TYPE "MEStoPLC_ResultsStoredScanExchange_ext"
VERSION : 0.1
   STRUCT
      Load_ResultsStored1OK : Bool;
      Load_ResultsStored1NG : Bool;
      Load_ResultsStored1ReqMesDone : Bool;
      Load_ResultsStored1Spare : Bool;
      Load_ResultsStored1Spare1 : Bool;
      Load_ResultsStored1Spare2 : Bool;
      Load_ResultsStored1Spare3 : Bool;
      Load_ResultsStored1Spare4 : Bool;
      Load_ResultsStored2OK : Bool;
      Load_ResultsStored2NG : Bool;
      Load_ResultsStored2ReqMesDone : Bool;
      Load_ResultsStored2Spare : Bool;
      Load_ResultsStored2Spare1 : Bool;
      Load_ResultsStored2Spare2 : Bool;
      Load_ResultsStored2Spare3 : Bool;
      Load_ResultsStored2Spare4 : Bool;
      Load_ResultsStored3OK : Bool;
      Load_ResultsStored3NG : Bool;
      Load_ResultsStored3ReqMesDone : Bool;
      Load_ResultsStored3Spare : Bool;
      Load_ResultsStored3Spare1 : Bool;
      Load_ResultsStored3Spare2 : Bool;
      Load_ResultsStored3Spare3 : Bool;
      Load_ResultsStored3Spare4 : Bool;
      Load_ResultsStored4OK : Bool;
      Load_ResultsStored4NG : Bool;
      Load_ResultsStored4ReqMesDone : Bool;
      Load_ResultsStored4Spare : Bool;
      Load_ResultsStored4Spare1 : Bool;
      Load_ResultsStored4Spare2 : Bool;
      Load_ResultsStored4Spare3 : Bool;
      Load_ResultsStored4Spare4 : Bool;
      Load_ResultsStored5OK : Bool;
      Load_ResultsStored5NG : Bool;
      Load_ResultsStored5ReqMesDone : Bool;
      Load_ResultsStored5Spare : Bool;
      Load_ResultsStored5Spare1 : Bool;
      Load_ResultsStored5Spare2 : Bool;
      Load_ResultsStored5Spare3 : Bool;
      Load_ResultsStored5Spare4 : Bool;
      Load_ResultsStored6OK : Bool;
      Load_ResultsStored6NG : Bool;
      Load_ResultsStored6ReqMesDone : Bool;
      Load_ResultsStored6Spare : Bool;
      Load_ResultsStored6Spare1 : Bool;
      Load_ResultsStored6Spare2 : Bool;
      Load_ResultsStored6Spare3 : Bool;
      Load_ResultsStored6Spare4 : Bool;
      Spare : Byte;
      Load_ResultsStored7OK : Bool;
      Load_ResultsStored7NG : Bool;
      Load_ResultsStored7ReqMesDone : Bool;
      Load_ResultsStored7Spare : Bool;
      Load_ResultsStored7Spare1 : Bool;
      Load_ResultsStored7Spare2 : Bool;
      Load_ResultsStored7Spare3 : Bool;
      Load_ResultsStored7Spare4 : Bool;
      Load_ResultsStored8OK : Bool;
      Load_ResultsStored8NG : Bool;
      Load_ResultsStored8ReqMesDone : Bool;
      Load_ResultsStored8Spare : Bool;
      Load_ResultsStored8Spare5 : Bool;
      Load_ResultsStored8Spare6 : Bool;
      Load_ResultsStored8Spare8 : Bool;
      Load_ResultsStored8Spare9 : Bool;
   END_STRUCT;

END_TYPE

